// TwinCAT 3 PLC project Sample
// ProgramVersion: 3.1.4020.2
// libraries:
//   Tc2_Standard, * (Beckhoff Automation GmbH)
//   Tc2_System, * (Beckhoff Automation GmbH)
//   Tc3_Module, * (Beckhoff Automation GmbH)
// project tree:
//   DUTs/ E_Foo01.TcDUT, E_Foo02.TcDUT
//   / PlcTask.TcTTO (not stored)
//   POUs/ MAIN.TcPOU
// real-time tasks:
//   TASK PlcTask: cycle T#10ms, priority 20, ADS port 350

// ---- DUTs/E_Foo01.TcDUT
{attribute 'qualified_only'}
TYPE E_Foo01 :
(
	eNoError := 0,
	eErrorA := 1,
	eErrorB := 2
);
END_TYPE

// ---- DUTs/E_Foo02.TcDUT
{attribute 'qualified_only'}
TYPE E_Foo02 :
(
	eNoError := 0,
	eError1 := 1,
	eError2 := 2
);
END_TYPE

// ---- POUs/MAIN.TcPOU
PROGRAM MAIN
VAR
	eFoo01		:	E_Foo01;
	eFoo02		:	E_Foo02;
END_VAR

eFoo01 := E_Foo01.eNoError;
eFoo02 := E_Foo02.eNoError;

END_PROGRAM
